// TIA Portal V19 export
DATA_BLOCK "PrjConfig_A03"   // DB82
// stored: MemoryReserve 100
   VAR
      Area03_Main : "AreaConfig";
   END_VAR
   VAR RETAIN
      A0301 : Struct
         Fermi_P1 : Struct
            Fermi : Array[1..6] of "ValveMachine_Config";
            Sfalsatore : "ValveMachine_Config";
            DelayMissingCondition : Time := T#3S;
         END_STRUCT;
         Fermi_P2 : Struct
            Fermi : Array[1..6] of "ValveMachine_Config";
            Sollevatori : Array[1..6] of "ValveMachine_Config";
            DelayMissingCondition : Time := T#3S;
         END_STRUCT;
         Fermi_P3 : Struct
            Fermi : Array[1..6] of "ValveMachine_Config";
            DelayMissingCondition : Time := T#3S;
         END_STRUCT;
         Fermi_P4 : Struct
            Fermi : Array[1..6] of "ValveMachine_Config";
            DelayMissingCondition : Time := T#3S;
         END_STRUCT;
         Trasporto { S7_SetPoint := 'True'} : "SpeedMachine_Config";
         Ribaltatore : Struct
            Ax : "Positioning_EPOS_Machine_Config_NEW";
            Solleva_Rib : Array[1..6] of "ValveMachine_Config";
         END_STRUCT;
         SpintoreLaterale : Struct
            Vrt_1 : "ValveMachine_Config";
            Orz_1 : "ValveMachine_Config";
            Vrt_2 : "ValveMachine_Config";
            Orz_2 : "ValveMachine_Config";
            Sollevatori : Array[1..7] of "ValveMachine_Config";
            QuotaIngombro_SpinLat2 : Real := 2680.0;
            QuotaIngombro_SpinLat1 { ExternalWritable := 'False'} : Real := 4777.0;
            DelayMissingCondition : Time := T#500MS;
         END_STRUCT;
      END_STRUCT;
      A0302 : Struct
         Spintore : Struct
            Ax : "Positioning_EPOS_Machine_Config_NEW";
            Vrt : "ValveMachine_Config";
            Orz : "ValveMachine_Config";
            SpintoreLat : Struct
               QuotaIngombro_SpinLat2 : Real := 2680.0;
               QuotaIngombro_SpinLat1 : Real := 4777.0;
            END_STRUCT;
            Bordatrice : Struct
               QuotaIngresso : Real := 801.0;
            END_STRUCT;
            DelayMissingCondition : Time := T#0MS;
         END_STRUCT;
         Bordatrice : Struct
            Ax : "Positioning_EPOS_Machine_Config_NEW";
            Measure : Struct
               K1_CarroPost : LReal := 674.0;   // K1: Misura tra carro di coda e sensore applicato per controllo ingombro pezzo con carro giù
               K2_BancoIngresso : LReal := 3560.0;   // K2: Misura interasse tra lo 0 al centro del banco e la FTC all'uscita della Bordatrice
            END_STRUCT;
         END_STRUCT;
         Regolaz_Bordatrice : Struct
            Formato : Struct
               Ax_D : Array[1..1] of "Positioning_DOL_Machine_Config";
               Ax_M : Array[1..10] of "Positioning_MOL_Machine_Config";
               M1_1 : "Positioning_DOL_Machine_Config";
               M1_2 : "Positioning_DOL_Machine_Config";
               M1_3 : "Positioning_MOL_Machine_Config";
               M1_4 : "Positioning_MOL_Machine_Config";
            END_STRUCT;
         END_STRUCT;
         Rulliera : Struct
            Ax : "SpeedMachine_Config";
         END_STRUCT;
         Centratori : Struct
            Centraggio : Array[1..3] of "ValveMachine_Config";
            Sollevamento : Array[1..3] of "ValveMachine_Config";
            DelayMissingCondition : Time := T#500MS;
            WorkWindows : Struct   // Finestre di disattivazione Centratore 1 e 3 in funzione dei Carri
               Coda : Struct
                  Min : LReal := 300.0;
                  Max : LReal := 1378.0;
               END_STRUCT;
               Testa : Struct
                  Min : LReal := 433.0;
                  Max : LReal := 970.0;
               END_STRUCT;
            END_STRUCT;
         END_STRUCT;
         PareggiatoreCoda : Struct
            Ax : "Positioning_DOL_Machine_Config";
            Bloccaggio : "ValveMachine_Config";
            BattutaVerticale : "ValveMachine_Config";
            PareggiatoreLong : "ValveMachine_Config";
            PosPareggiatore : Struct
               QuotaMin_Work : LReal := 82.0;
               QuotaMax_Work { S7_SetPoint := 'True'} : LReal := 91.0;
            END_STRUCT;
            MinDistanzaConSpalla { S7_SetPoint := 'True'} : LReal := 85.7;
            DelayMissingCondition : Time := T#200MS;
         END_STRUCT;
         PareggiatoreTesta : Struct
            Ax : "Positioning_DOL_Machine_Config";
            Bloccaggio : "ValveMachine_Config";
            Sollevamento : "ValveMachine_Config";
            Centraggio : "ValveMachine_Config";
            MinDistanzaConSpalla : LReal := 5.0;
            DelayMissingCondition : Time := T#200MS;
         END_STRUCT;
         Manipolatore : Struct
            Testa : Struct
               Ax : "Positioning_EPOS_Machine_Config_NEW";
               Sollevatore : "ValveMachine_Config";
               Magnete : "ValveMachine_Config";
            END_STRUCT;
            Coda : Struct
               Ax : "Positioning_EPOS_Machine_Config_NEW";
               Sollevatore : "ValveMachine_Config";
               Magnete : "ValveMachine_Config";
            END_STRUCT;
            DelayMissingCondition : Time := T#200MS;
         END_STRUCT;
      END_STRUCT;
   END_VAR
BEGIN
   Area03_Main.TimeOutStopImmediate := T#1S_500MS;
   Area03_Main.TimeOutStopInPhase := T#10S;
   Area03_Main.TimeOutStopProgrammed := T#5M;
   Area03_Main.TimeOutResetAlarms := T#1S;
   A0301.Fermi_P1.Fermi[1..6].DelayPressureRunningTimeout := T#3S;
   A0301.Fermi_P1.Fermi[1..6].DelayMissingCondition := T#3S;
   A0301.Fermi_P1.Fermi[1..6].Rest_LsQty := 1;
   A0301.Fermi_P1.Fermi[1..6].Work_LsQty := 0;
   A0301.Fermi_P1.Fermi[1..6].Rest_RetainAut := FALSE;
   A0301.Fermi_P1.Fermi[1..6].Work_RetainAut := FALSE;
   A0301.Fermi_P1.Fermi[1..6].V.RestLimSwitchExist := TRUE;
   A0301.Fermi_P1.Fermi[1..6].V.WorkLimSwitchExist := FALSE;
   A0301.Fermi_P1.Fermi[1..6].V.CheckOilInPressure := FALSE;
   A0301.Fermi_P1.Fermi[1..6].V.CutRestWhenIsAtRest := TRUE;
   A0301.Fermi_P1.Fermi[1..6].V.CutWorkWhenIsAtWork := FALSE;
   A0301.Fermi_P1.Fermi[1..6].V.RestTime := T#1MS;
   A0301.Fermi_P1.Fermi[1..6].V.WorkTime := T#100MS;
   A0301.Fermi_P1.Fermi[1..6].V.RestTimeOut := T#4S;
   A0301.Fermi_P1.Fermi[1..6].V.WorkTimeOut := T#4S;
   A0301.Fermi_P1.Sfalsatore.DelayPressureRunningTimeout := T#3S;
   A0301.Fermi_P1.Sfalsatore.DelayMissingCondition := T#3S;
   A0301.Fermi_P1.Sfalsatore.Rest_LsQty := 1;
   A0301.Fermi_P1.Sfalsatore.Work_LsQty := 1;
   A0301.Fermi_P1.Sfalsatore.Rest_RetainAut := FALSE;
   A0301.Fermi_P1.Sfalsatore.Work_RetainAut := FALSE;
   A0301.Fermi_P1.Sfalsatore.V.RestLimSwitchExist := TRUE;
   A0301.Fermi_P1.Sfalsatore.V.WorkLimSwitchExist := TRUE;
   A0301.Fermi_P1.Sfalsatore.V.CheckOilInPressure := FALSE;
   A0301.Fermi_P1.Sfalsatore.V.CutRestWhenIsAtRest := FALSE;
   A0301.Fermi_P1.Sfalsatore.V.CutWorkWhenIsAtWork := TRUE;
   A0301.Fermi_P1.Sfalsatore.V.RestTime := T#1S;
   A0301.Fermi_P1.Sfalsatore.V.WorkTime := T#300MS;
   A0301.Fermi_P1.Sfalsatore.V.RestTimeOut := T#1H;
   A0301.Fermi_P1.Sfalsatore.V.WorkTimeOut := T#1H;
   A0301.Fermi_P2.Fermi[1..6].DelayPressureRunningTimeout := T#3S;
   A0301.Fermi_P2.Fermi[1..6].DelayMissingCondition := T#3S;
   A0301.Fermi_P2.Fermi[1..6].Rest_LsQty := 1;
   A0301.Fermi_P2.Fermi[1..6].Work_LsQty := 0;
   A0301.Fermi_P2.Fermi[1..6].Rest_RetainAut := FALSE;
   A0301.Fermi_P2.Fermi[1..6].Work_RetainAut := FALSE;
   A0301.Fermi_P2.Fermi[1..6].V.RestLimSwitchExist := TRUE;
   A0301.Fermi_P2.Fermi[1..6].V.WorkLimSwitchExist := FALSE;
   A0301.Fermi_P2.Fermi[1..6].V.CheckOilInPressure := FALSE;
   A0301.Fermi_P2.Fermi[1..6].V.CutRestWhenIsAtRest := TRUE;
   A0301.Fermi_P2.Fermi[1..6].V.CutWorkWhenIsAtWork := FALSE;
   A0301.Fermi_P2.Fermi[1..6].V.RestTime := T#1MS;
   A0301.Fermi_P2.Fermi[1..6].V.WorkTime := T#100MS;
   A0301.Fermi_P2.Fermi[1..6].V.RestTimeOut := T#4S;
   A0301.Fermi_P2.Fermi[1..6].V.WorkTimeOut := T#4S;
   A0301.Fermi_P2.Sollevatori[1..6].DelayPressureRunningTimeout := T#3S;
   A0301.Fermi_P2.Sollevatori[1..6].DelayMissingCondition := T#3S;
   A0301.Fermi_P2.Sollevatori[1..6].Rest_LsQty := 1;
   A0301.Fermi_P2.Sollevatori[1..6].Work_LsQty := 0;
   A0301.Fermi_P2.Sollevatori[1..6].Rest_RetainAut := FALSE;
   A0301.Fermi_P2.Sollevatori[1..6].Work_RetainAut := FALSE;
   A0301.Fermi_P2.Sollevatori[1..6].V.RestLimSwitchExist := TRUE;
   A0301.Fermi_P2.Sollevatori[1..6].V.WorkLimSwitchExist := FALSE;
   A0301.Fermi_P2.Sollevatori[1..6].V.CheckOilInPressure := FALSE;
   A0301.Fermi_P2.Sollevatori[1..6].V.CutRestWhenIsAtRest := TRUE;
   A0301.Fermi_P2.Sollevatori[1..6].V.CutWorkWhenIsAtWork := FALSE;
   A0301.Fermi_P2.Sollevatori[1..6].V.RestTime := T#1MS;
   A0301.Fermi_P2.Sollevatori[1..6].V.WorkTime := T#100MS;
   A0301.Fermi_P2.Sollevatori[1..6].V.RestTimeOut := T#4S;
   A0301.Fermi_P2.Sollevatori[1..6].V.WorkTimeOut := T#4S;
   A0301.Fermi_P3.Fermi[1..6].DelayPressureRunningTimeout := T#3S;
   A0301.Fermi_P3.Fermi[1..6].DelayMissingCondition := T#3S;
   A0301.Fermi_P3.Fermi[1..6].Rest_LsQty := 1;
   A0301.Fermi_P3.Fermi[1..6].Work_LsQty := 0;
   A0301.Fermi_P3.Fermi[1..6].Rest_RetainAut := FALSE;
   A0301.Fermi_P3.Fermi[1..6].Work_RetainAut := FALSE;
   A0301.Fermi_P3.Fermi[1..6].V.RestLimSwitchExist := TRUE;
   A0301.Fermi_P3.Fermi[1..6].V.WorkLimSwitchExist := FALSE;
   A0301.Fermi_P3.Fermi[1..6].V.CheckOilInPressure := FALSE;
   A0301.Fermi_P3.Fermi[1..6].V.CutRestWhenIsAtRest := TRUE;
   A0301.Fermi_P3.Fermi[1..6].V.CutWorkWhenIsAtWork := FALSE;
   A0301.Fermi_P3.Fermi[1..6].V.RestTime := T#1MS;
   A0301.Fermi_P3.Fermi[1..6].V.WorkTime := T#100MS;
   A0301.Fermi_P3.Fermi[1..6].V.RestTimeOut := T#4S;
   A0301.Fermi_P3.Fermi[1..6].V.WorkTimeOut := T#4S;
   A0301.Fermi_P4.Fermi[1..6].DelayPressureRunningTimeout := T#3S;
   A0301.Fermi_P4.Fermi[1..6].DelayMissingCondition := T#3S;
   A0301.Fermi_P4.Fermi[1..6].Rest_LsQty := 1;
   A0301.Fermi_P4.Fermi[1..6].Work_LsQty := 0;
   A0301.Fermi_P4.Fermi[1..6].Rest_RetainAut := FALSE;
   A0301.Fermi_P4.Fermi[1..6].Work_RetainAut := FALSE;
   A0301.Fermi_P4.Fermi[1..6].V.RestLimSwitchExist := TRUE;
   A0301.Fermi_P4.Fermi[1..6].V.WorkLimSwitchExist := FALSE;
   A0301.Fermi_P4.Fermi[1..6].V.CheckOilInPressure := FALSE;
   A0301.Fermi_P4.Fermi[1..6].V.CutRestWhenIsAtRest := TRUE;
   A0301.Fermi_P4.Fermi[1..6].V.CutWorkWhenIsAtWork := FALSE;
   A0301.Fermi_P4.Fermi[1..6].V.RestTime := T#1MS;
   A0301.Fermi_P4.Fermi[1..6].V.WorkTime := T#300MS;
   A0301.Fermi_P4.Fermi[1..6].V.RestTimeOut := T#4S;
   A0301.Fermi_P4.Fermi[1..6].V.WorkTimeOut := T#4S;
   A0301.Trasporto.SLS_VEL := 5000.0;
   A0301.Trasporto.DelayMissingCondition := T#3S;
   A0301.Trasporto.Ax.SINA_Drive.ReferenceVelocity := 2200.0;
   A0301.Trasporto.Ax.SINA_Drive.InvertDirection := FALSE;
   A0301.Trasporto.Ax.MinAccTime := 0.1;
   A0301.Trasporto.Ax.MinDecTime := 0.1;
   A0301.Trasporto.Ax.LeadScrewPitchVal := 359.8;
   A0301.Trasporto.Ax.MotorRevolution := 20.0;
   A0301.Trasporto.Ax.LoadRevolution := 1.0;
   A0301.Trasporto.Ax.PowerOffDelay := T#1S_500MS;
   A0301.Trasporto.Ax.StandstillVelocity := 50.0;
   A0301.Trasporto.Ax.StandstillDelay := T#100MS;
   A0301.Trasporto.Fan.Presence := FALSE;
   A0301.Trasporto.Fan.DelayOff := T#0MS;
   A0301.Trasporto.Brake_Presence := FALSE;
   A0301.Ribaltatore.Ax.SLS_Vel := 3000.0;
   A0301.Ribaltatore.Ax.DelayMissingCondition := T#100MS;
   A0301.Ribaltatore.Ax.Ax.Encoder_Inc_AutoReloadPosition := FALSE;
   A0301.Ribaltatore.Ax.Ax.Encoder_is_Absolute := TRUE;
   A0301.Ribaltatore.Ax.Ax.LeadScrewPitchVal := 9.0000015;
   A0301.Ribaltatore.Ax.Ax.MotorRevolution := 23.33;
   A0301.Ribaltatore.Ax.Ax.LoadRevolution := 1.0;
   A0301.Ribaltatore.Ax.Ax.PowerOffDelay := T#100MS;
   A0301.Ribaltatore.Ax.Ax.MaxRPM_S120_P2000 := 3000.0;
   A0301.Ribaltatore.Ax.Ax.MaxVel_S120_P2571 := 6000.0;
   A0301.Ribaltatore.Ax.Ax.MaxAcc_S120_P2572 := 50.0;
   A0301.Ribaltatore.Ax.Ax.MaxDec_S120_P2573 := 50.0;
   A0301.Ribaltatore.Ax.Ax.Modulo_S120_P2566 := 0.0;
   A0301.Ribaltatore.Ax.Ax.SwLimMinus_S120_P2580 := 0.25;
   A0301.Ribaltatore.Ax.Ax.SwLimPlus_S120_P2581 := 125.0;
   A0301.Ribaltatore.Ax.Fan.Presence := FALSE;
   A0301.Ribaltatore.Ax.Fan.DelayOff := T#0MS;
   A0301.Ribaltatore.Ax.Brake_Presence := FALSE;
   A0301.Ribaltatore.Solleva_Rib[1..6].DelayPressureRunningTimeout := T#3S;
   A0301.Ribaltatore.Solleva_Rib[1..6].DelayMissingCondition := T#3S;
   A0301.Ribaltatore.Solleva_Rib[1..6].Rest_LsQty := 1;
   A0301.Ribaltatore.Solleva_Rib[1..6].Work_LsQty := 1;
   A0301.Ribaltatore.Solleva_Rib[1..6].Rest_RetainAut := FALSE;
   A0301.Ribaltatore.Solleva_Rib[1..6].Work_RetainAut := FALSE;
   A0301.Ribaltatore.Solleva_Rib[1..6].V.RestLimSwitchExist := TRUE;
   A0301.Ribaltatore.Solleva_Rib[1..6].V.WorkLimSwitchExist := TRUE;
   A0301.Ribaltatore.Solleva_Rib[1..6].V.CheckOilInPressure := FALSE;
   A0301.Ribaltatore.Solleva_Rib[1..6].V.CutRestWhenIsAtRest := FALSE;
   A0301.Ribaltatore.Solleva_Rib[1..6].V.CutWorkWhenIsAtWork := FALSE;
   A0301.Ribaltatore.Solleva_Rib[1..6].V.RestTime := T#1MS;
   A0301.Ribaltatore.Solleva_Rib[1..6].V.WorkTime := T#200MS;
   A0301.Ribaltatore.Solleva_Rib[1..6].V.RestTimeOut := T#5S;
   A0301.Ribaltatore.Solleva_Rib[1..6].V.WorkTimeOut := T#5S;
   A0301.SpintoreLaterale.Vrt_1.DelayPressureRunningTimeout := T#3S;
   A0301.SpintoreLaterale.Vrt_1.DelayMissingCondition := T#3S;
   A0301.SpintoreLaterale.Vrt_1.Rest_LsQty := 1;
   A0301.SpintoreLaterale.Vrt_1.Work_LsQty := 0;
   A0301.SpintoreLaterale.Vrt_1.Rest_RetainAut := FALSE;
   A0301.SpintoreLaterale.Vrt_1.Work_RetainAut := FALSE;
   A0301.SpintoreLaterale.Vrt_1.V.RestLimSwitchExist := TRUE;
   A0301.SpintoreLaterale.Vrt_1.V.WorkLimSwitchExist := FALSE;
   A0301.SpintoreLaterale.Vrt_1.V.CheckOilInPressure := FALSE;
   A0301.SpintoreLaterale.Vrt_1.V.CutRestWhenIsAtRest := TRUE;
   A0301.SpintoreLaterale.Vrt_1.V.CutWorkWhenIsAtWork := FALSE;
   A0301.SpintoreLaterale.Vrt_1.V.RestTime := T#1MS;
   A0301.SpintoreLaterale.Vrt_1.V.WorkTime := T#300MS;
   A0301.SpintoreLaterale.Vrt_1.V.RestTimeOut := T#5S;
   A0301.SpintoreLaterale.Vrt_1.V.WorkTimeOut := T#5S;
   A0301.SpintoreLaterale.Orz_1.DelayPressureRunningTimeout := T#3S;
   A0301.SpintoreLaterale.Orz_1.DelayMissingCondition := T#3S;
   A0301.SpintoreLaterale.Orz_1.Rest_LsQty := 1;
   A0301.SpintoreLaterale.Orz_1.Work_LsQty := 0;
   A0301.SpintoreLaterale.Orz_1.Rest_RetainAut := FALSE;
   A0301.SpintoreLaterale.Orz_1.Work_RetainAut := FALSE;
   A0301.SpintoreLaterale.Orz_1.V.RestLimSwitchExist := TRUE;
   A0301.SpintoreLaterale.Orz_1.V.WorkLimSwitchExist := FALSE;
   A0301.SpintoreLaterale.Orz_1.V.CheckOilInPressure := FALSE;
   A0301.SpintoreLaterale.Orz_1.V.CutRestWhenIsAtRest := FALSE;
   A0301.SpintoreLaterale.Orz_1.V.CutWorkWhenIsAtWork := FALSE;
   A0301.SpintoreLaterale.Orz_1.V.RestTime := T#1MS;
   A0301.SpintoreLaterale.Orz_1.V.WorkTime := T#300MS;
   A0301.SpintoreLaterale.Orz_1.V.RestTimeOut := T#5S;
   A0301.SpintoreLaterale.Orz_1.V.WorkTimeOut := T#5S;
   A0301.SpintoreLaterale.Vrt_2.DelayPressureRunningTimeout := T#3S;
   A0301.SpintoreLaterale.Vrt_2.DelayMissingCondition := T#3S;
   A0301.SpintoreLaterale.Vrt_2.Rest_LsQty := 1;
   A0301.SpintoreLaterale.Vrt_2.Work_LsQty := 0;
   A0301.SpintoreLaterale.Vrt_2.Rest_RetainAut := FALSE;
   A0301.SpintoreLaterale.Vrt_2.Work_RetainAut := FALSE;
   A0301.SpintoreLaterale.Vrt_2.V.RestLimSwitchExist := TRUE;
   A0301.SpintoreLaterale.Vrt_2.V.WorkLimSwitchExist := FALSE;
   A0301.SpintoreLaterale.Vrt_2.V.CheckOilInPressure := FALSE;
   A0301.SpintoreLaterale.Vrt_2.V.CutRestWhenIsAtRest := TRUE;
   A0301.SpintoreLaterale.Vrt_2.V.CutWorkWhenIsAtWork := FALSE;
   A0301.SpintoreLaterale.Vrt_2.V.RestTime := T#1MS;
   A0301.SpintoreLaterale.Vrt_2.V.WorkTime := T#300MS;
   A0301.SpintoreLaterale.Vrt_2.V.RestTimeOut := T#5S;
   A0301.SpintoreLaterale.Vrt_2.V.WorkTimeOut := T#5S;
   A0301.SpintoreLaterale.Orz_2.DelayPressureRunningTimeout := T#3S;
   A0301.SpintoreLaterale.Orz_2.DelayMissingCondition := T#3S;
   A0301.SpintoreLaterale.Orz_2.Rest_LsQty := 1;
   A0301.SpintoreLaterale.Orz_2.Work_LsQty := 0;
   A0301.SpintoreLaterale.Orz_2.Rest_RetainAut := FALSE;
   A0301.SpintoreLaterale.Orz_2.Work_RetainAut := FALSE;
   A0301.SpintoreLaterale.Orz_2.V.RestLimSwitchExist := TRUE;
   A0301.SpintoreLaterale.Orz_2.V.WorkLimSwitchExist := FALSE;
   A0301.SpintoreLaterale.Orz_2.V.CheckOilInPressure := FALSE;
   A0301.SpintoreLaterale.Orz_2.V.CutRestWhenIsAtRest := FALSE;
   A0301.SpintoreLaterale.Orz_2.V.CutWorkWhenIsAtWork := FALSE;
   A0301.SpintoreLaterale.Orz_2.V.RestTime := T#1MS;
   A0301.SpintoreLaterale.Orz_2.V.WorkTime := T#300MS;
   A0301.SpintoreLaterale.Orz_2.V.RestTimeOut := T#5S;
   A0301.SpintoreLaterale.Orz_2.V.WorkTimeOut := T#5S;
   A0301.SpintoreLaterale.Sollevatori[1..7].DelayPressureRunningTimeout := T#3S;
   A0301.SpintoreLaterale.Sollevatori[1..7].DelayMissingCondition := T#3S;
   A0301.SpintoreLaterale.Sollevatori[1..7].Rest_LsQty := 1;
   A0301.SpintoreLaterale.Sollevatori[1..7].Work_LsQty := 0;
   A0301.SpintoreLaterale.Sollevatori[1..7].Rest_RetainAut := FALSE;
   A0301.SpintoreLaterale.Sollevatori[1..7].Work_RetainAut := FALSE;
   A0301.SpintoreLaterale.Sollevatori[1..7].V.RestLimSwitchExist := TRUE;
   A0301.SpintoreLaterale.Sollevatori[1..7].V.WorkLimSwitchExist := FALSE;
   A0301.SpintoreLaterale.Sollevatori[1..7].V.CheckOilInPressure := FALSE;
   A0301.SpintoreLaterale.Sollevatori[1..7].V.CutRestWhenIsAtRest := TRUE;
   A0301.SpintoreLaterale.Sollevatori[1..7].V.CutWorkWhenIsAtWork := TRUE;
   A0301.SpintoreLaterale.Sollevatori[1..7].V.RestTime := T#1S;
   A0301.SpintoreLaterale.Sollevatori[1..7].V.WorkTime := T#500MS;
   A0301.SpintoreLaterale.Sollevatori[1..7].V.RestTimeOut := T#4S;
   A0301.SpintoreLaterale.Sollevatori[1..7].V.WorkTimeOut := T#4S;
   A0302.Spintore.Ax.SLS_Vel := 3000.0;
   A0302.Spintore.Ax.DelayMissingCondition := T#1S;
   A0302.Spintore.Ax.Ax.Encoder_Inc_AutoReloadPosition := FALSE;
   A0302.Spintore.Ax.Ax.Encoder_is_Absolute := TRUE;
   A0302.Spintore.Ax.Ax.LeadScrewPitchVal := 287.989799;
   A0302.Spintore.Ax.Ax.MotorRevolution := 10.0;
   A0302.Spintore.Ax.Ax.LoadRevolution := 1.0;
   A0302.Spintore.Ax.Ax.PowerOffDelay := T#1S;
   A0302.Spintore.Ax.Ax.MaxRPM_S120_P2000 := 3000.0;
   A0302.Spintore.Ax.Ax.MaxVel_S120_P2571 := 86396.0;
   A0302.Spintore.Ax.Ax.MaxAcc_S120_P2572 := 5000.0;
   A0302.Spintore.Ax.Ax.MaxDec_S120_P2573 := 5000.0;
   A0302.Spintore.Ax.Ax.Modulo_S120_P2566 := 0.0;
   A0302.Spintore.Ax.Ax.SwLimMinus_S120_P2580 := 0.5;
   A0302.Spintore.Ax.Ax.SwLimPlus_S120_P2581 := 5370.0;
   A0302.Spintore.Ax.Fan.Presence := FALSE;
   A0302.Spintore.Ax.Fan.DelayOff := T#0MS;
   A0302.Spintore.Ax.Brake_Presence := FALSE;
   A0302.Spintore.Vrt.DelayPressureRunningTimeout := T#3S;
   A0302.Spintore.Vrt.DelayMissingCondition := T#3S;
   A0302.Spintore.Vrt.Rest_LsQty := 1;
   A0302.Spintore.Vrt.Work_LsQty := 1;
   A0302.Spintore.Vrt.Rest_RetainAut := FALSE;
   A0302.Spintore.Vrt.Work_RetainAut := FALSE;
   A0302.Spintore.Vrt.V.RestLimSwitchExist := TRUE;
   A0302.Spintore.Vrt.V.WorkLimSwitchExist := TRUE;
   A0302.Spintore.Vrt.V.CheckOilInPressure := FALSE;
   A0302.Spintore.Vrt.V.CutRestWhenIsAtRest := TRUE;
   A0302.Spintore.Vrt.V.CutWorkWhenIsAtWork := FALSE;
   A0302.Spintore.Vrt.V.RestTime := T#10MS;
   A0302.Spintore.Vrt.V.WorkTime := T#100MS;
   A0302.Spintore.Vrt.V.RestTimeOut := T#4S;
   A0302.Spintore.Vrt.V.WorkTimeOut := T#4S;
   A0302.Spintore.Orz.DelayPressureRunningTimeout := T#3S;
   A0302.Spintore.Orz.DelayMissingCondition := T#3S;
   A0302.Spintore.Orz.Rest_LsQty := 1;
   A0302.Spintore.Orz.Work_LsQty := 0;
   A0302.Spintore.Orz.Rest_RetainAut := FALSE;
   A0302.Spintore.Orz.Work_RetainAut := FALSE;
   A0302.Spintore.Orz.V.RestLimSwitchExist := TRUE;
   A0302.Spintore.Orz.V.WorkLimSwitchExist := FALSE;
   A0302.Spintore.Orz.V.CheckOilInPressure := FALSE;
   A0302.Spintore.Orz.V.CutRestWhenIsAtRest := TRUE;
   A0302.Spintore.Orz.V.CutWorkWhenIsAtWork := FALSE;
   A0302.Spintore.Orz.V.RestTime := T#10MS;
   A0302.Spintore.Orz.V.WorkTime := T#100MS;
   A0302.Spintore.Orz.V.RestTimeOut := T#4S;
   A0302.Spintore.Orz.V.WorkTimeOut := T#4S;
   A0302.Bordatrice.Ax.SLS_Vel := 3000.0;
   A0302.Bordatrice.Ax.DelayMissingCondition := T#200MS;
   A0302.Bordatrice.Ax.Ax.Encoder_Inc_AutoReloadPosition := TRUE;
   A0302.Bordatrice.Ax.Ax.Encoder_is_Absolute := FALSE;
   A0302.Bordatrice.Ax.Ax.LeadScrewPitchVal := 486.946;
   A0302.Bordatrice.Ax.Ax.MotorRevolution := 12.4;
   A0302.Bordatrice.Ax.Ax.LoadRevolution := 1.0;
   A0302.Bordatrice.Ax.Ax.PowerOffDelay := T#500MS;
   A0302.Bordatrice.Ax.Ax.MaxRPM_S120_P2000 := 3000.0;
   A0302.Bordatrice.Ax.Ax.MaxVel_S120_P2571 := 60000.0;
   A0302.Bordatrice.Ax.Ax.MaxAcc_S120_P2572 := 4000.0;
   A0302.Bordatrice.Ax.Ax.MaxDec_S120_P2573 := 4000.0;
   A0302.Bordatrice.Ax.Ax.Modulo_S120_P2566 := 1000000000.0;
   A0302.Bordatrice.Ax.Ax.SwLimMinus_S120_P2580 := 0.0;
   A0302.Bordatrice.Ax.Ax.SwLimPlus_S120_P2581 := 0.0;
   A0302.Bordatrice.Ax.Fan.Presence := FALSE;
   A0302.Bordatrice.Ax.Fan.DelayOff := T#0MS;
   A0302.Bordatrice.Ax.Brake_Presence := FALSE;
   A0302.Regolaz_Bordatrice.Formato.Ax_D[1].DelayMissingCondition := T#3S;
   A0302.Regolaz_Bordatrice.Formato.Ax_D[1].CyclicOBTime_ms := 10.0;
   A0302.Regolaz_Bordatrice.Formato.Ax_D[1].Ax.limitMinus := 59.0;
   A0302.Regolaz_Bordatrice.Formato.Ax_D[1].Ax.limitPlus := 215.0;
   A0302.Regolaz_Bordatrice.Formato.Ax_D[1].Ax.Backlash := 0.4;
   A0302.Regolaz_Bordatrice.Formato.Ax_D[1].Ax.BacklashActivation := TRUE;
   A0302.Regolaz_Bordatrice.Formato.Ax_D[1].Ax.ToleranceWindow := 0.0;
   A0302.Regolaz_Bordatrice.Formato.Ax_D[1].Ax.ToleranceWindowDelay := T#100MS;
   A0302.Regolaz_Bordatrice.Formato.Ax_D[1].Ax.PreCutOff := 0.03;
   A0302.Regolaz_Bordatrice.Formato.Ax_D[1].Ax.PreEndLowSpeed := 0.0;
   A0302.Regolaz_Bordatrice.Formato.Ax_D[1].Ax.PreEndMedSpeed := 0.0;
   A0302.Regolaz_Bordatrice.Formato.Ax_D[1].Ax.ChangeDirectionDelay := T#0MS;
   A0302.Regolaz_Bordatrice.Formato.Ax_D[1].Ax.StandstillVelocity := 0.5;
   A0302.Regolaz_Bordatrice.Formato.Ax_D[1].Ax.StandStillDelay := T#100MS;
   A0302.Regolaz_Bordatrice.Formato.Ax_D[1].Ax.HomingDirection := FALSE;
   A0302.Regolaz_Bordatrice.Formato.Ax_D[1].Ax.RecallTime := 0.0;
   A0302.Regolaz_Bordatrice.Formato.Ax_D[1].Ax.VelocityFilter_T := 10.0;
   A0302.Regolaz_Bordatrice.Formato.Ax_D[1].Ax.VelocityMeasUnit := 2;
   A0302.Regolaz_Bordatrice.Formato.Ax_D[1].Ax.PosFbkDisabled := FALSE;
   A0302.Regolaz_Bordatrice.Formato.Ax_D[1].Ax.FbkCtrlDisabled := TRUE;
   A0302.Regolaz_Bordatrice.Formato.Ax_D[1].Ax_UM2."m" := -1.0;
   A0302.Regolaz_Bordatrice.Formato.Ax_D[1].Ax_UM2.q := 320.5;
   A0302.Regolaz_Bordatrice.Formato.Ax_D[1].S120.SpeedMotor.ReferenceVelocity := 2200.0;
   A0302.Regolaz_Bordatrice.Formato.Ax_D[1].S120.SpeedMotor.InvertDirection := FALSE;
   A0302.Regolaz_Bordatrice.Formato.Ax_D[1].S120.PowerOffDelay := T#1S_500MS;
   A0302.Regolaz_Bordatrice.Formato.Ax_D[1].S120.StandstillVelocity := 20.0;
   A0302.Regolaz_Bordatrice.Formato.Ax_D[1].S120.AccTime := 0.5;
   A0302.Regolaz_Bordatrice.Formato.Ax_D[1].S120.DecTime := 0.5;
   A0302.Regolaz_Bordatrice.Formato.Ax_D[1].Fan.Presence := FALSE;
   A0302.Regolaz_Bordatrice.Formato.Ax_D[1].Fan.DelayOff := T#10M;
   A0302.Regolaz_Bordatrice.Formato.Ax_D[1].Brake_Presence := FALSE;
   A0302.Regolaz_Bordatrice.Formato.Ax_M[1..10].DelayMissingCondition := T#100MS;
   A0302.Regolaz_Bordatrice.Formato.Ax_M[1..10].CyclicOBTime_ms := 10.0;
   A0302.Regolaz_Bordatrice.Formato.Ax_M[1..10].Ax.limitMinus := 38.0;
   A0302.Regolaz_Bordatrice.Formato.Ax_M[1..10].Ax.limitPlus := 52.0;
   A0302.Regolaz_Bordatrice.Formato.Ax_M[1..10].Ax.Backlash := 0.4;
   A0302.Regolaz_Bordatrice.Formato.Ax_M[1..10].Ax.BacklashActivation := TRUE;
   A0302.Regolaz_Bordatrice.Formato.Ax_M[1..10].Ax.ToleranceWindow := 0.0;
   A0302.Regolaz_Bordatrice.Formato.Ax_M[1..10].Ax.ToleranceWindowDelay := T#100MS;
   A0302.Regolaz_Bordatrice.Formato.Ax_M[1..10].Ax.PreCutOff := 0.03;
   A0302.Regolaz_Bordatrice.Formato.Ax_M[1..10].Ax.PreEndLowSpeed := 0.0;
   A0302.Regolaz_Bordatrice.Formato.Ax_M[1..10].Ax.PreEndMedSpeed := 0.0;
   A0302.Regolaz_Bordatrice.Formato.Ax_M[1..10].Ax.ChangeDirectionDelay := T#0MS;
   A0302.Regolaz_Bordatrice.Formato.Ax_M[1..10].Ax.StandstillVelocity := 0.5;
   A0302.Regolaz_Bordatrice.Formato.Ax_M[1..10].Ax.StandStillDelay := T#100MS;
   A0302.Regolaz_Bordatrice.Formato.Ax_M[1..10].Ax.HomingDirection := FALSE;
   A0302.Regolaz_Bordatrice.Formato.Ax_M[1..10].Ax.RecallTime := 0.0;
   A0302.Regolaz_Bordatrice.Formato.Ax_M[1..10].Ax.VelocityFilter_T := 10.0;
   A0302.Regolaz_Bordatrice.Formato.Ax_M[1..10].Ax.VelocityMeasUnit := 2;
   A0302.Regolaz_Bordatrice.Formato.Ax_M[1..10].Ax.PosFbkDisabled := FALSE;
   A0302.Regolaz_Bordatrice.Formato.Ax_M[1..10].Ax.FbkCtrlDisabled := TRUE;
   A0302.Regolaz_Bordatrice.Formato.Ax_M[1..10].Ax_UM2."m" := 1.0;
   A0302.Regolaz_Bordatrice.Formato.Ax_M[1..5].Ax_UM2.q := 127.0;
   A0302.Regolaz_Bordatrice.Formato.Ax_M[6..10].Ax_UM2.q := 84.8;
   A0302.Regolaz_Bordatrice.Formato.M1_1.DelayMissingCondition := T#3S;
   A0302.Regolaz_Bordatrice.Formato.M1_1.CyclicOBTime_ms := 10.0;
   A0302.Regolaz_Bordatrice.Formato.M1_1.Ax.limitMinus := 0.0;
   A0302.Regolaz_Bordatrice.Formato.M1_1.Ax.limitPlus := 0.0;
   A0302.Regolaz_Bordatrice.Formato.M1_1.Ax.Backlash := 0.0;
   A0302.Regolaz_Bordatrice.Formato.M1_1.Ax.BacklashActivation := FALSE;
   A0302.Regolaz_Bordatrice.Formato.M1_1.Ax.ToleranceWindow := 0.0;
   A0302.Regolaz_Bordatrice.Formato.M1_1.Ax.ToleranceWindowDelay := T#0MS;
   A0302.Regolaz_Bordatrice.Formato.M1_1.Ax.PreCutOff := 0.0;
   A0302.Regolaz_Bordatrice.Formato.M1_1.Ax.PreEndLowSpeed := 0.0;
   A0302.Regolaz_Bordatrice.Formato.M1_1.Ax.PreEndMedSpeed := 0.0;
   A0302.Regolaz_Bordatrice.Formato.M1_1.Ax.ChangeDirectionDelay := T#0MS;
   A0302.Regolaz_Bordatrice.Formato.M1_1.Ax.StandstillVelocity := 0.0;
   A0302.Regolaz_Bordatrice.Formato.M1_1.Ax.StandStillDelay := T#0MS;
   A0302.Regolaz_Bordatrice.Formato.M1_1.Ax.HomingDirection := FALSE;
   A0302.Regolaz_Bordatrice.Formato.M1_1.Ax.RecallTime := 0.0;
   A0302.Regolaz_Bordatrice.Formato.M1_1.Ax.VelocityFilter_T := 10.0;
   A0302.Regolaz_Bordatrice.Formato.M1_1.Ax.VelocityMeasUnit := 0;
   A0302.Regolaz_Bordatrice.Formato.M1_1.Ax.PosFbkDisabled := FALSE;
   A0302.Regolaz_Bordatrice.Formato.M1_1.Ax.FbkCtrlDisabled := FALSE;
   A0302.Regolaz_Bordatrice.Formato.M1_1.Ax_UM2."m" := 1.0;
   A0302.Regolaz_Bordatrice.Formato.M1_1.Ax_UM2.q := 0.0;
   A0302.Regolaz_Bordatrice.Formato.M1_1.S120.SpeedMotor.ReferenceVelocity := 2000.0;
   A0302.Regolaz_Bordatrice.Formato.M1_1.S120.SpeedMotor.InvertDirection := FALSE;
   A0302.Regolaz_Bordatrice.Formato.M1_1.S120.PowerOffDelay := T#1S_500MS;
   A0302.Regolaz_Bordatrice.Formato.M1_1.S120.StandstillVelocity := 0.0;
   A0302.Regolaz_Bordatrice.Formato.M1_1.S120.AccTime := 0.0;
   A0302.Regolaz_Bordatrice.Formato.M1_1.S120.DecTime := 0.0;
   A0302.Regolaz_Bordatrice.Formato.M1_1.Fan.Presence := FALSE;
   A0302.Regolaz_Bordatrice.Formato.M1_1.Fan.DelayOff := T#10M;
   A0302.Regolaz_Bordatrice.Formato.M1_1.Brake_Presence := FALSE;
   A0302.Regolaz_Bordatrice.Formato.M1_2.DelayMissingCondition := T#3S;
   A0302.Regolaz_Bordatrice.Formato.M1_2.CyclicOBTime_ms := 10.0;
   A0302.Regolaz_Bordatrice.Formato.M1_2.Ax.limitMinus := 0.0;
   A0302.Regolaz_Bordatrice.Formato.M1_2.Ax.limitPlus := 0.0;
   A0302.Regolaz_Bordatrice.Formato.M1_2.Ax.Backlash := 0.0;
   A0302.Regolaz_Bordatrice.Formato.M1_2.Ax.BacklashActivation := FALSE;
   A0302.Regolaz_Bordatrice.Formato.M1_2.Ax.ToleranceWindow := 0.0;
   A0302.Regolaz_Bordatrice.Formato.M1_2.Ax.ToleranceWindowDelay := T#0MS;
   A0302.Regolaz_Bordatrice.Formato.M1_2.Ax.PreCutOff := 0.0;
   A0302.Regolaz_Bordatrice.Formato.M1_2.Ax.PreEndLowSpeed := 0.0;
   A0302.Regolaz_Bordatrice.Formato.M1_2.Ax.PreEndMedSpeed := 0.0;
   A0302.Regolaz_Bordatrice.Formato.M1_2.Ax.ChangeDirectionDelay := T#0MS;
   A0302.Regolaz_Bordatrice.Formato.M1_2.Ax.StandstillVelocity := 0.0;
   A0302.Regolaz_Bordatrice.Formato.M1_2.Ax.StandStillDelay := T#0MS;
   A0302.Regolaz_Bordatrice.Formato.M1_2.Ax.HomingDirection := FALSE;
   A0302.Regolaz_Bordatrice.Formato.M1_2.Ax.RecallTime := 0.0;
   A0302.Regolaz_Bordatrice.Formato.M1_2.Ax.VelocityFilter_T := 10.0;
   A0302.Regolaz_Bordatrice.Formato.M1_2.Ax.VelocityMeasUnit := 0;
   A0302.Regolaz_Bordatrice.Formato.M1_2.Ax.PosFbkDisabled := FALSE;
   A0302.Regolaz_Bordatrice.Formato.M1_2.Ax.FbkCtrlDisabled := FALSE;
   A0302.Regolaz_Bordatrice.Formato.M1_2.Ax_UM2."m" := 1.0;
   A0302.Regolaz_Bordatrice.Formato.M1_2.Ax_UM2.q := 0.0;
   A0302.Regolaz_Bordatrice.Formato.M1_2.S120.SpeedMotor.ReferenceVelocity := 2000.0;
   A0302.Regolaz_Bordatrice.Formato.M1_2.S120.SpeedMotor.InvertDirection := FALSE;
   A0302.Regolaz_Bordatrice.Formato.M1_2.S120.PowerOffDelay := T#1S_500MS;
   A0302.Regolaz_Bordatrice.Formato.M1_2.S120.StandstillVelocity := 0.0;
   A0302.Regolaz_Bordatrice.Formato.M1_2.S120.AccTime := 0.0;
   A0302.Regolaz_Bordatrice.Formato.M1_2.S120.DecTime := 0.0;
   A0302.Regolaz_Bordatrice.Formato.M1_2.Fan.Presence := FALSE;
   A0302.Regolaz_Bordatrice.Formato.M1_2.Fan.DelayOff := T#10M;
   A0302.Regolaz_Bordatrice.Formato.M1_2.Brake_Presence := FALSE;
   A0302.Regolaz_Bordatrice.Formato.M1_3.DelayMissingCondition := T#0MS;
   A0302.Regolaz_Bordatrice.Formato.M1_3.CyclicOBTime_ms := 0.0;
   A0302.Regolaz_Bordatrice.Formato.M1_3.Ax.limitMinus := 0.0;
   A0302.Regolaz_Bordatrice.Formato.M1_3.Ax.limitPlus := 0.0;
   A0302.Regolaz_Bordatrice.Formato.M1_3.Ax.Backlash := 0.0;
   A0302.Regolaz_Bordatrice.Formato.M1_3.Ax.BacklashActivation := FALSE;
   A0302.Regolaz_Bordatrice.Formato.M1_3.Ax.ToleranceWindow := 0.0;
   A0302.Regolaz_Bordatrice.Formato.M1_3.Ax.ToleranceWindowDelay := T#0MS;
   A0302.Regolaz_Bordatrice.Formato.M1_3.Ax.PreCutOff := 0.0;
   A0302.Regolaz_Bordatrice.Formato.M1_3.Ax.PreEndLowSpeed := 0.0;
   A0302.Regolaz_Bordatrice.Formato.M1_3.Ax.PreEndMedSpeed := 0.0;
   A0302.Regolaz_Bordatrice.Formato.M1_3.Ax.ChangeDirectionDelay := T#0MS;
   A0302.Regolaz_Bordatrice.Formato.M1_3.Ax.StandstillVelocity := 0.0;
   A0302.Regolaz_Bordatrice.Formato.M1_3.Ax.StandStillDelay := T#0MS;
   A0302.Regolaz_Bordatrice.Formato.M1_3.Ax.HomingDirection := FALSE;
   A0302.Regolaz_Bordatrice.Formato.M1_3.Ax.RecallTime := 0.0;
   A0302.Regolaz_Bordatrice.Formato.M1_3.Ax.VelocityFilter_T := 10.0;
   A0302.Regolaz_Bordatrice.Formato.M1_3.Ax.VelocityMeasUnit := 0;
   A0302.Regolaz_Bordatrice.Formato.M1_3.Ax.PosFbkDisabled := FALSE;
   A0302.Regolaz_Bordatrice.Formato.M1_3.Ax.FbkCtrlDisabled := FALSE;
   A0302.Regolaz_Bordatrice.Formato.M1_3.Ax_UM2."m" := 0.0;
   A0302.Regolaz_Bordatrice.Formato.M1_3.Ax_UM2.q := 0.0;
   A0302.Regolaz_Bordatrice.Formato.M1_4.DelayMissingCondition := T#0MS;
   A0302.Regolaz_Bordatrice.Formato.M1_4.CyclicOBTime_ms := 0.0;
   A0302.Regolaz_Bordatrice.Formato.M1_4.Ax.limitMinus := 0.0;
   A0302.Regolaz_Bordatrice.Formato.M1_4.Ax.limitPlus := 0.0;
   A0302.Regolaz_Bordatrice.Formato.M1_4.Ax.Backlash := 0.0;
   A0302.Regolaz_Bordatrice.Formato.M1_4.Ax.BacklashActivation := FALSE;
   A0302.Regolaz_Bordatrice.Formato.M1_4.Ax.ToleranceWindow := 0.0;
   A0302.Regolaz_Bordatrice.Formato.M1_4.Ax.ToleranceWindowDelay := T#0MS;
   A0302.Regolaz_Bordatrice.Formato.M1_4.Ax.PreCutOff := 0.0;
   A0302.Regolaz_Bordatrice.Formato.M1_4.Ax.PreEndLowSpeed := 0.0;
   A0302.Regolaz_Bordatrice.Formato.M1_4.Ax.PreEndMedSpeed := 0.0;
   A0302.Regolaz_Bordatrice.Formato.M1_4.Ax.ChangeDirectionDelay := T#0MS;
   A0302.Regolaz_Bordatrice.Formato.M1_4.Ax.StandstillVelocity := 0.0;
   A0302.Regolaz_Bordatrice.Formato.M1_4.Ax.StandStillDelay := T#0MS;
   A0302.Regolaz_Bordatrice.Formato.M1_4.Ax.HomingDirection := FALSE;
   A0302.Regolaz_Bordatrice.Formato.M1_4.Ax.RecallTime := 0.0;
   A0302.Regolaz_Bordatrice.Formato.M1_4.Ax.VelocityFilter_T := 10.0;
   A0302.Regolaz_Bordatrice.Formato.M1_4.Ax.VelocityMeasUnit := 0;
   A0302.Regolaz_Bordatrice.Formato.M1_4.Ax.PosFbkDisabled := FALSE;
   A0302.Regolaz_Bordatrice.Formato.M1_4.Ax.FbkCtrlDisabled := FALSE;
   A0302.Regolaz_Bordatrice.Formato.M1_4.Ax_UM2."m" := 0.0;
   A0302.Regolaz_Bordatrice.Formato.M1_4.Ax_UM2.q := 0.0;
   A0302.Rulliera.Ax.SLS_VEL := 3000.0;
   A0302.Rulliera.Ax.DelayMissingCondition := T#3S;
   A0302.Rulliera.Ax.Ax.SINA_Drive.ReferenceVelocity := 2200.0;
   A0302.Rulliera.Ax.Ax.SINA_Drive.InvertDirection := FALSE;
   A0302.Rulliera.Ax.Ax.MinAccTime := 0.1;
   A0302.Rulliera.Ax.Ax.MinDecTime := 0.1;
   A0302.Rulliera.Ax.Ax.LeadScrewPitchVal := 219.91;   // 359.98
   A0302.Rulliera.Ax.Ax.MotorRevolution := 6.364;
   A0302.Rulliera.Ax.Ax.LoadRevolution := 1.0;
   A0302.Rulliera.Ax.Ax.PowerOffDelay := T#1S_500MS;
   A0302.Rulliera.Ax.Ax.StandstillVelocity := 50.0;
   A0302.Rulliera.Ax.Ax.StandstillDelay := T#100MS;
   A0302.Rulliera.Ax.Fan.Presence := FALSE;
   A0302.Rulliera.Ax.Fan.DelayOff := T#0MS;
   A0302.Rulliera.Ax.Brake_Presence := FALSE;
   A0302.Centratori.Centraggio[1..3].DelayPressureRunningTimeout := T#3S;
   A0302.Centratori.Centraggio[1..3].DelayMissingCondition := T#3S;
   A0302.Centratori.Centraggio[1..3].Rest_LsQty := 1;
   A0302.Centratori.Centraggio[1..3].Work_LsQty := 0;
   A0302.Centratori.Centraggio[1..3].Rest_RetainAut := FALSE;
   A0302.Centratori.Centraggio[1..3].Work_RetainAut := FALSE;
   A0302.Centratori.Centraggio[1..3].V.RestLimSwitchExist := TRUE;
   A0302.Centratori.Centraggio[1..3].V.WorkLimSwitchExist := FALSE;
   A0302.Centratori.Centraggio[1..3].V.CheckOilInPressure := FALSE;
   A0302.Centratori.Centraggio[1..3].V.CutRestWhenIsAtRest := TRUE;
   A0302.Centratori.Centraggio[1..3].V.CutWorkWhenIsAtWork := FALSE;
   A0302.Centratori.Centraggio[1..3].V.RestTime := T#10MS;
   A0302.Centratori.Centraggio[1..3].V.WorkTime := T#300MS;
   A0302.Centratori.Centraggio[1..3].V.RestTimeOut := T#4S;
   A0302.Centratori.Centraggio[1..3].V.WorkTimeOut := T#4S;
   A0302.Centratori.Sollevamento[1..3].DelayPressureRunningTimeout := T#3S;
   A0302.Centratori.Sollevamento[1..3].DelayMissingCondition := T#3S;
   A0302.Centratori.Sollevamento[1..3].Rest_LsQty := 1;
   A0302.Centratori.Sollevamento[1..3].Work_LsQty := 1;
   A0302.Centratori.Sollevamento[1..3].Rest_RetainAut := FALSE;
   A0302.Centratori.Sollevamento[1..3].Work_RetainAut := FALSE;
   A0302.Centratori.Sollevamento[1..3].V.RestLimSwitchExist := TRUE;
   A0302.Centratori.Sollevamento[1..3].V.WorkLimSwitchExist := TRUE;
   A0302.Centratori.Sollevamento[1..3].V.CheckOilInPressure := FALSE;
   A0302.Centratori.Sollevamento[1..3].V.CutRestWhenIsAtRest := TRUE;
   A0302.Centratori.Sollevamento[1..3].V.CutWorkWhenIsAtWork := FALSE;
   A0302.Centratori.Sollevamento[1..3].V.RestTime := T#10MS;
   A0302.Centratori.Sollevamento[1..3].V.WorkTime := T#10MS;
   A0302.Centratori.Sollevamento[1..3].V.RestTimeOut := T#4S;
   A0302.Centratori.Sollevamento[1..3].V.WorkTimeOut := T#4S;
   A0302.PareggiatoreCoda.Ax.DelayMissingCondition := T#3S;
   A0302.PareggiatoreCoda.Ax.CyclicOBTime_ms := 10.0;
   A0302.PareggiatoreCoda.Ax.Ax.limitMinus := 430.0;
   A0302.PareggiatoreCoda.Ax.Ax.limitPlus := 2870.0;
   A0302.PareggiatoreCoda.Ax.Ax.Backlash := 0.0;
   A0302.PareggiatoreCoda.Ax.Ax.BacklashActivation := FALSE;
   A0302.PareggiatoreCoda.Ax.Ax.ToleranceWindow := 0.1;
   A0302.PareggiatoreCoda.Ax.Ax.ToleranceWindowDelay := T#100MS;
   A0302.PareggiatoreCoda.Ax.Ax.PreCutOff := 0.0;
   A0302.PareggiatoreCoda.Ax.Ax.PreEndLowSpeed := 0.0;
   A0302.PareggiatoreCoda.Ax.Ax.PreEndMedSpeed := 0.0;
   A0302.PareggiatoreCoda.Ax.Ax.ChangeDirectionDelay := T#0MS;
   A0302.PareggiatoreCoda.Ax.Ax.StandstillVelocity := 0.5;
   A0302.PareggiatoreCoda.Ax.Ax.StandStillDelay := T#100MS;
   A0302.PareggiatoreCoda.Ax.Ax.HomingDirection := FALSE;
   A0302.PareggiatoreCoda.Ax.Ax.RecallTime := 0.0;
   A0302.PareggiatoreCoda.Ax.Ax.VelocityFilter_T := 10.0;
   A0302.PareggiatoreCoda.Ax.Ax.VelocityMeasUnit := 2;
   A0302.PareggiatoreCoda.Ax.Ax.PosFbkDisabled := FALSE;
   A0302.PareggiatoreCoda.Ax.Ax.FbkCtrlDisabled := TRUE;
   A0302.PareggiatoreCoda.Ax.Ax_UM2."m" := 1.0;
   A0302.PareggiatoreCoda.Ax.Ax_UM2.q := -433.0;
   A0302.PareggiatoreCoda.Ax.S120.SpeedMotor.ReferenceVelocity := 2000.0;
   A0302.PareggiatoreCoda.Ax.S120.SpeedMotor.InvertDirection := FALSE;
   A0302.PareggiatoreCoda.Ax.S120.PowerOffDelay := T#5S;
   A0302.PareggiatoreCoda.Ax.S120.StandstillVelocity := 50.0;
   A0302.PareggiatoreCoda.Ax.S120.AccTime := 0.5;
   A0302.PareggiatoreCoda.Ax.S120.DecTime := 0.5;
   A0302.PareggiatoreCoda.Ax.Fan.Presence := FALSE;
   A0302.PareggiatoreCoda.Ax.Fan.DelayOff := T#10M;
   A0302.PareggiatoreCoda.Ax.Brake_Presence := FALSE;
   A0302.PareggiatoreCoda.Bloccaggio.DelayPressureRunningTimeout := T#3S;
   A0302.PareggiatoreCoda.Bloccaggio.DelayMissingCondition := T#3S;
   A0302.PareggiatoreCoda.Bloccaggio.Rest_LsQty := 1;
   A0302.PareggiatoreCoda.Bloccaggio.Work_LsQty := 1;
   A0302.PareggiatoreCoda.Bloccaggio.Rest_RetainAut := FALSE;
   A0302.PareggiatoreCoda.Bloccaggio.Work_RetainAut := FALSE;
   A0302.PareggiatoreCoda.Bloccaggio.V.RestLimSwitchExist := TRUE;
   A0302.PareggiatoreCoda.Bloccaggio.V.WorkLimSwitchExist := TRUE;
   A0302.PareggiatoreCoda.Bloccaggio.V.CheckOilInPressure := TRUE;
   A0302.PareggiatoreCoda.Bloccaggio.V.CutRestWhenIsAtRest := FALSE;
   A0302.PareggiatoreCoda.Bloccaggio.V.CutWorkWhenIsAtWork := FALSE;
   A0302.PareggiatoreCoda.Bloccaggio.V.RestTime := T#500MS;
   A0302.PareggiatoreCoda.Bloccaggio.V.WorkTime := T#500MS;
   A0302.PareggiatoreCoda.Bloccaggio.V.RestTimeOut := T#4S;
   A0302.PareggiatoreCoda.Bloccaggio.V.WorkTimeOut := T#4S;
   A0302.PareggiatoreCoda.BattutaVerticale.DelayPressureRunningTimeout := T#3S;
   A0302.PareggiatoreCoda.BattutaVerticale.DelayMissingCondition := T#3S;
   A0302.PareggiatoreCoda.BattutaVerticale.Rest_LsQty := 1;
   A0302.PareggiatoreCoda.BattutaVerticale.Work_LsQty := 1;
   A0302.PareggiatoreCoda.BattutaVerticale.Rest_RetainAut := FALSE;
   A0302.PareggiatoreCoda.BattutaVerticale.Work_RetainAut := FALSE;
   A0302.PareggiatoreCoda.BattutaVerticale.V.RestLimSwitchExist := TRUE;
   A0302.PareggiatoreCoda.BattutaVerticale.V.WorkLimSwitchExist := TRUE;
   A0302.PareggiatoreCoda.BattutaVerticale.V.CheckOilInPressure := FALSE;
   A0302.PareggiatoreCoda.BattutaVerticale.V.CutRestWhenIsAtRest := FALSE;
   A0302.PareggiatoreCoda.BattutaVerticale.V.CutWorkWhenIsAtWork := FALSE;
   A0302.PareggiatoreCoda.BattutaVerticale.V.RestTime := T#1MS;
   A0302.PareggiatoreCoda.BattutaVerticale.V.WorkTime := T#50MS;
   A0302.PareggiatoreCoda.BattutaVerticale.V.RestTimeOut := T#3S;
   A0302.PareggiatoreCoda.BattutaVerticale.V.WorkTimeOut := T#3S;
   A0302.PareggiatoreCoda.PareggiatoreLong.DelayPressureRunningTimeout := T#3S;
   A0302.PareggiatoreCoda.PareggiatoreLong.DelayMissingCondition := T#3S;
   A0302.PareggiatoreCoda.PareggiatoreLong.Rest_LsQty := 1;
   A0302.PareggiatoreCoda.PareggiatoreLong.Work_LsQty := 1;
   A0302.PareggiatoreCoda.PareggiatoreLong.Rest_RetainAut := FALSE;
   A0302.PareggiatoreCoda.PareggiatoreLong.Work_RetainAut := FALSE;
   A0302.PareggiatoreCoda.PareggiatoreLong.V.RestLimSwitchExist := TRUE;
   A0302.PareggiatoreCoda.PareggiatoreLong.V.WorkLimSwitchExist := TRUE;
   A0302.PareggiatoreCoda.PareggiatoreLong.V.CheckOilInPressure := TRUE;
   A0302.PareggiatoreCoda.PareggiatoreLong.V.CutRestWhenIsAtRest := TRUE;
   A0302.PareggiatoreCoda.PareggiatoreLong.V.CutWorkWhenIsAtWork := FALSE;
   A0302.PareggiatoreCoda.PareggiatoreLong.V.RestTime := T#500MS;
   A0302.PareggiatoreCoda.PareggiatoreLong.V.WorkTime := T#5S;
   A0302.PareggiatoreCoda.PareggiatoreLong.V.RestTimeOut := T#4S;
   A0302.PareggiatoreCoda.PareggiatoreLong.V.WorkTimeOut := T#7S;
   A0302.PareggiatoreTesta.Ax.DelayMissingCondition := T#3S;
   A0302.PareggiatoreTesta.Ax.CyclicOBTime_ms := 10.0;
   A0302.PareggiatoreTesta.Ax.Ax.limitMinus := 87.0;
   A0302.PareggiatoreTesta.Ax.Ax.limitPlus := 2502.0;
   A0302.PareggiatoreTesta.Ax.Ax.Backlash := 0.0;
   A0302.PareggiatoreTesta.Ax.Ax.BacklashActivation := FALSE;
   A0302.PareggiatoreTesta.Ax.Ax.ToleranceWindow := 0.1;
   A0302.PareggiatoreTesta.Ax.Ax.ToleranceWindowDelay := T#100MS;
   A0302.PareggiatoreTesta.Ax.Ax.PreCutOff := 0.0;
   A0302.PareggiatoreTesta.Ax.Ax.PreEndLowSpeed := 0.0;
   A0302.PareggiatoreTesta.Ax.Ax.PreEndMedSpeed := 0.0;
   A0302.PareggiatoreTesta.Ax.Ax.ChangeDirectionDelay := T#0MS;
   A0302.PareggiatoreTesta.Ax.Ax.StandstillVelocity := 0.5;
   A0302.PareggiatoreTesta.Ax.Ax.StandStillDelay := T#100MS;
   A0302.PareggiatoreTesta.Ax.Ax.HomingDirection := FALSE;
   A0302.PareggiatoreTesta.Ax.Ax.RecallTime := 0.0;
   A0302.PareggiatoreTesta.Ax.Ax.VelocityFilter_T := 10.0;
   A0302.PareggiatoreTesta.Ax.Ax.VelocityMeasUnit := 2;
   A0302.PareggiatoreTesta.Ax.Ax.PosFbkDisabled := FALSE;
   A0302.PareggiatoreTesta.Ax.Ax.FbkCtrlDisabled := TRUE;
   A0302.PareggiatoreTesta.Ax.Ax_UM2."m" := 1.0;
   A0302.PareggiatoreTesta.Ax.Ax_UM2.q := -343.0;
   A0302.PareggiatoreTesta.Ax.S120.SpeedMotor.ReferenceVelocity := 2000.0;
   A0302.PareggiatoreTesta.Ax.S120.SpeedMotor.InvertDirection := FALSE;
   A0302.PareggiatoreTesta.Ax.S120.PowerOffDelay := T#5S;
   A0302.PareggiatoreTesta.Ax.S120.StandstillVelocity := 50.0;
   A0302.PareggiatoreTesta.Ax.S120.AccTime := 0.25;
   A0302.PareggiatoreTesta.Ax.S120.DecTime := 0.25;
   A0302.PareggiatoreTesta.Ax.Fan.Presence := FALSE;
   A0302.PareggiatoreTesta.Ax.Fan.DelayOff := T#10M;
   A0302.PareggiatoreTesta.Ax.Brake_Presence := FALSE;
   A0302.PareggiatoreTesta.Bloccaggio.DelayPressureRunningTimeout := T#3S;
   A0302.PareggiatoreTesta.Bloccaggio.DelayMissingCondition := T#3S;
   A0302.PareggiatoreTesta.Bloccaggio.Rest_LsQty := 1;
   A0302.PareggiatoreTesta.Bloccaggio.Work_LsQty := 1;
   A0302.PareggiatoreTesta.Bloccaggio.Rest_RetainAut := FALSE;
   A0302.PareggiatoreTesta.Bloccaggio.Work_RetainAut := FALSE;
   A0302.PareggiatoreTesta.Bloccaggio.V.RestLimSwitchExist := TRUE;
   A0302.PareggiatoreTesta.Bloccaggio.V.WorkLimSwitchExist := TRUE;
   A0302.PareggiatoreTesta.Bloccaggio.V.CheckOilInPressure := TRUE;
   A0302.PareggiatoreTesta.Bloccaggio.V.CutRestWhenIsAtRest := FALSE;
   A0302.PareggiatoreTesta.Bloccaggio.V.CutWorkWhenIsAtWork := FALSE;
   A0302.PareggiatoreTesta.Bloccaggio.V.RestTime := T#500MS;
   A0302.PareggiatoreTesta.Bloccaggio.V.WorkTime := T#500MS;
   A0302.PareggiatoreTesta.Bloccaggio.V.RestTimeOut := T#4S;
   A0302.PareggiatoreTesta.Bloccaggio.V.WorkTimeOut := T#4S;
   A0302.PareggiatoreTesta.Sollevamento.DelayPressureRunningTimeout := T#3S;
   A0302.PareggiatoreTesta.Sollevamento.DelayMissingCondition := T#3S;
   A0302.PareggiatoreTesta.Sollevamento.Rest_LsQty := 1;
   A0302.PareggiatoreTesta.Sollevamento.Work_LsQty := 1;
   A0302.PareggiatoreTesta.Sollevamento.Rest_RetainAut := FALSE;
   A0302.PareggiatoreTesta.Sollevamento.Work_RetainAut := FALSE;
   A0302.PareggiatoreTesta.Sollevamento.V.RestLimSwitchExist := TRUE;
   A0302.PareggiatoreTesta.Sollevamento.V.WorkLimSwitchExist := TRUE;
   A0302.PareggiatoreTesta.Sollevamento.V.CheckOilInPressure := FALSE;
   A0302.PareggiatoreTesta.Sollevamento.V.CutRestWhenIsAtRest := FALSE;
   A0302.PareggiatoreTesta.Sollevamento.V.CutWorkWhenIsAtWork := FALSE;
   A0302.PareggiatoreTesta.Sollevamento.V.RestTime := T#10MS;
   A0302.PareggiatoreTesta.Sollevamento.V.WorkTime := T#10MS;
   A0302.PareggiatoreTesta.Sollevamento.V.RestTimeOut := T#5S;
   A0302.PareggiatoreTesta.Sollevamento.V.WorkTimeOut := T#5S;
   A0302.PareggiatoreTesta.Centraggio.DelayPressureRunningTimeout := T#3S;
   A0302.PareggiatoreTesta.Centraggio.DelayMissingCondition := T#3S;
   A0302.PareggiatoreTesta.Centraggio.Rest_LsQty := 1;
   A0302.PareggiatoreTesta.Centraggio.Work_LsQty := 1;
   A0302.PareggiatoreTesta.Centraggio.Rest_RetainAut := FALSE;
   A0302.PareggiatoreTesta.Centraggio.Work_RetainAut := FALSE;
   A0302.PareggiatoreTesta.Centraggio.V.RestLimSwitchExist := TRUE;
   A0302.PareggiatoreTesta.Centraggio.V.WorkLimSwitchExist := FALSE;
   A0302.PareggiatoreTesta.Centraggio.V.CheckOilInPressure := FALSE;
   A0302.PareggiatoreTesta.Centraggio.V.CutRestWhenIsAtRest := FALSE;
   A0302.PareggiatoreTesta.Centraggio.V.CutWorkWhenIsAtWork := FALSE;
   A0302.PareggiatoreTesta.Centraggio.V.RestTime := T#10MS;
   A0302.PareggiatoreTesta.Centraggio.V.WorkTime := T#10MS;
   A0302.PareggiatoreTesta.Centraggio.V.RestTimeOut := T#5S;
   A0302.PareggiatoreTesta.Centraggio.V.WorkTimeOut := T#5S;
   A0302.Manipolatore.Testa.Ax.SLS_Vel := 3000.0;
   A0302.Manipolatore.Testa.Ax.DelayMissingCondition := T#1S;
   A0302.Manipolatore.Testa.Ax.Ax.Encoder_Inc_AutoReloadPosition := FALSE;
   A0302.Manipolatore.Testa.Ax.Ax.Encoder_is_Absolute := TRUE;
   A0302.Manipolatore.Testa.Ax.Ax.LeadScrewPitchVal := 10.4992026;
   A0302.Manipolatore.Testa.Ax.Ax.MotorRevolution := 66.84;
   A0302.Manipolatore.Testa.Ax.Ax.LoadRevolution := 1.0;
   A0302.Manipolatore.Testa.Ax.Ax.PowerOffDelay := T#500MS;
   A0302.Manipolatore.Testa.Ax.Ax.MaxRPM_S120_P2000 := 8000.0;
   A0302.Manipolatore.Testa.Ax.Ax.MaxVel_S120_P2571 := 31500.0;
   A0302.Manipolatore.Testa.Ax.Ax.MaxAcc_S120_P2572 := 2000.0;
   A0302.Manipolatore.Testa.Ax.Ax.MaxDec_S120_P2573 := 2000.0;
   A0302.Manipolatore.Testa.Ax.Ax.Modulo_S120_P2566 := 0.0;
   A0302.Manipolatore.Testa.Ax.Ax.SwLimMinus_S120_P2580 := -650.0;
   A0302.Manipolatore.Testa.Ax.Ax.SwLimPlus_S120_P2581 := 553.0;
   A0302.Manipolatore.Testa.Ax.Fan.Presence := FALSE;
   A0302.Manipolatore.Testa.Ax.Fan.DelayOff := T#0MS;
   A0302.Manipolatore.Testa.Ax.Brake_Presence := FALSE;
   A0302.Manipolatore.Testa.Sollevatore.DelayPressureRunningTimeout := T#3S;
   A0302.Manipolatore.Testa.Sollevatore.DelayMissingCondition := T#3S;
   A0302.Manipolatore.Testa.Sollevatore.Rest_LsQty := 1;
   A0302.Manipolatore.Testa.Sollevatore.Work_LsQty := 0;
   A0302.Manipolatore.Testa.Sollevatore.Rest_RetainAut := FALSE;
   A0302.Manipolatore.Testa.Sollevatore.Work_RetainAut := FALSE;
   A0302.Manipolatore.Testa.Sollevatore.V.RestLimSwitchExist := TRUE;
   A0302.Manipolatore.Testa.Sollevatore.V.WorkLimSwitchExist := FALSE;
   A0302.Manipolatore.Testa.Sollevatore.V.CheckOilInPressure := FALSE;
   A0302.Manipolatore.Testa.Sollevatore.V.CutRestWhenIsAtRest := FALSE;
   A0302.Manipolatore.Testa.Sollevatore.V.CutWorkWhenIsAtWork := FALSE;
   A0302.Manipolatore.Testa.Sollevatore.V.RestTime := T#1MS;
   A0302.Manipolatore.Testa.Sollevatore.V.WorkTime := T#200MS;
   A0302.Manipolatore.Testa.Sollevatore.V.RestTimeOut := T#5S;
   A0302.Manipolatore.Testa.Sollevatore.V.WorkTimeOut := T#5S;
   A0302.Manipolatore.Testa.Magnete.DelayPressureRunningTimeout := T#3S;
   A0302.Manipolatore.Testa.Magnete.DelayMissingCondition := T#3S;
   A0302.Manipolatore.Testa.Magnete.Rest_LsQty := 1;
   A0302.Manipolatore.Testa.Magnete.Work_LsQty := 0;
   A0302.Manipolatore.Testa.Magnete.Rest_RetainAut := FALSE;
   A0302.Manipolatore.Testa.Magnete.Work_RetainAut := FALSE;
   A0302.Manipolatore.Testa.Magnete.V.RestLimSwitchExist := TRUE;
   A0302.Manipolatore.Testa.Magnete.V.WorkLimSwitchExist := FALSE;
   A0302.Manipolatore.Testa.Magnete.V.CheckOilInPressure := FALSE;
   A0302.Manipolatore.Testa.Magnete.V.CutRestWhenIsAtRest := TRUE;
   A0302.Manipolatore.Testa.Magnete.V.CutWorkWhenIsAtWork := FALSE;
   A0302.Manipolatore.Testa.Magnete.V.RestTime := T#1MS;
   A0302.Manipolatore.Testa.Magnete.V.WorkTime := T#300MS;
   A0302.Manipolatore.Testa.Magnete.V.RestTimeOut := T#5S;
   A0302.Manipolatore.Testa.Magnete.V.WorkTimeOut := T#5S;
   A0302.Manipolatore.Coda.Ax.SLS_Vel := 3000.0;
   A0302.Manipolatore.Coda.Ax.DelayMissingCondition := T#1S;
   A0302.Manipolatore.Coda.Ax.Ax.Encoder_Inc_AutoReloadPosition := FALSE;
   A0302.Manipolatore.Coda.Ax.Ax.Encoder_is_Absolute := TRUE;
   A0302.Manipolatore.Coda.Ax.Ax.LeadScrewPitchVal := 10.4992026;
   A0302.Manipolatore.Coda.Ax.Ax.MotorRevolution := 66.84;
   A0302.Manipolatore.Coda.Ax.Ax.LoadRevolution := 0.0;
   A0302.Manipolatore.Coda.Ax.Ax.PowerOffDelay := T#0MS;
   A0302.Manipolatore.Coda.Ax.Ax.MaxRPM_S120_P2000 := 8000.0;
   A0302.Manipolatore.Coda.Ax.Ax.MaxVel_S120_P2571 := 31500.0;
   A0302.Manipolatore.Coda.Ax.Ax.MaxAcc_S120_P2572 := 2000.0;
   A0302.Manipolatore.Coda.Ax.Ax.MaxDec_S120_P2573 := 2000.0;
   A0302.Manipolatore.Coda.Ax.Ax.Modulo_S120_P2566 := 0.0;
   A0302.Manipolatore.Coda.Ax.Ax.SwLimMinus_S120_P2580 := -650.0;
   A0302.Manipolatore.Coda.Ax.Ax.SwLimPlus_S120_P2581 := 552.0;
   A0302.Manipolatore.Coda.Ax.Fan.Presence := FALSE;
   A0302.Manipolatore.Coda.Ax.Fan.DelayOff := T#0MS;
   A0302.Manipolatore.Coda.Ax.Brake_Presence := FALSE;
   A0302.Manipolatore.Coda.Sollevatore.DelayPressureRunningTimeout := T#3S;
   A0302.Manipolatore.Coda.Sollevatore.DelayMissingCondition := T#3S;
   A0302.Manipolatore.Coda.Sollevatore.Rest_LsQty := 1;
   A0302.Manipolatore.Coda.Sollevatore.Work_LsQty := 0;
   A0302.Manipolatore.Coda.Sollevatore.Rest_RetainAut := FALSE;
   A0302.Manipolatore.Coda.Sollevatore.Work_RetainAut := FALSE;
   A0302.Manipolatore.Coda.Sollevatore.V.RestLimSwitchExist := TRUE;
   A0302.Manipolatore.Coda.Sollevatore.V.WorkLimSwitchExist := FALSE;
   A0302.Manipolatore.Coda.Sollevatore.V.CheckOilInPressure := FALSE;
   A0302.Manipolatore.Coda.Sollevatore.V.CutRestWhenIsAtRest := FALSE;
   A0302.Manipolatore.Coda.Sollevatore.V.CutWorkWhenIsAtWork := FALSE;
   A0302.Manipolatore.Coda.Sollevatore.V.RestTime := T#1MS;
   A0302.Manipolatore.Coda.Sollevatore.V.WorkTime := T#200MS;
   A0302.Manipolatore.Coda.Sollevatore.V.RestTimeOut := T#5S;
   A0302.Manipolatore.Coda.Sollevatore.V.WorkTimeOut := T#5S;
   A0302.Manipolatore.Coda.Magnete.DelayPressureRunningTimeout := T#3S;
   A0302.Manipolatore.Coda.Magnete.DelayMissingCondition := T#3S;
   A0302.Manipolatore.Coda.Magnete.Rest_LsQty := 1;
   A0302.Manipolatore.Coda.Magnete.Work_LsQty := 0;
   A0302.Manipolatore.Coda.Magnete.Rest_RetainAut := FALSE;
   A0302.Manipolatore.Coda.Magnete.Work_RetainAut := FALSE;
   A0302.Manipolatore.Coda.Magnete.V.RestLimSwitchExist := TRUE;
   A0302.Manipolatore.Coda.Magnete.V.WorkLimSwitchExist := FALSE;
   A0302.Manipolatore.Coda.Magnete.V.CheckOilInPressure := FALSE;
   A0302.Manipolatore.Coda.Magnete.V.CutRestWhenIsAtRest := TRUE;
   A0302.Manipolatore.Coda.Magnete.V.CutWorkWhenIsAtWork := FALSE;
   A0302.Manipolatore.Coda.Magnete.V.RestTime := T#1MS;
   A0302.Manipolatore.Coda.Magnete.V.WorkTime := T#300MS;
   A0302.Manipolatore.Coda.Magnete.V.RestTimeOut := T#5S;
   A0302.Manipolatore.Coda.Magnete.V.WorkTimeOut := T#5S;
END_DATA_BLOCK
